FUNCTION_BLOCK PLC01A1 (* Access IOs of the PLC01A1 module *)
  (* Standard: 61499-2; Description: Copyright (c) 2019 fortiss GmbH This program and the accompanying materials are made available under the terms of the Eclipse Public License 2.0 which is available at https://www.eclipse.org/legal/epl-2.0/ SPDX-License-Identifier: EPL-2.0 *)
  (* Version 1.0, 2019-10-01, Jose Cabral, fortiss GmbH *)
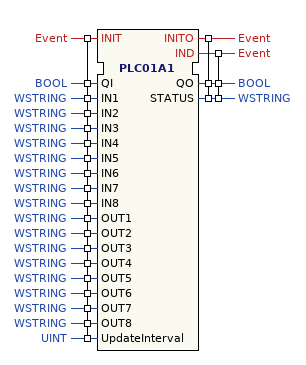
  EVENT_INPUT
    INIT WITH QI, UpdateInterval, IN1, IN2, IN3, IN4, IN5, IN6, IN7, IN8, OUT1, OUT2, OUT3, OUT4, OUT5, OUT6, OUT7, OUT8; (* Service Initialization *)
  END_EVENT
  EVENT_OUTPUT
    INITO WITH QO, STATUS; (* Initialization Confirm *)
    IND WITH QO, STATUS; (* Indication from Resource *)
  END_EVENT
  VAR_INPUT
    QI : BOOL; (* Event Input Qualifier *)
    IN1 : WSTRING;
    IN2 : WSTRING;
    IN3 : WSTRING;
    IN4 : WSTRING;
    IN5 : WSTRING;
    IN6 : WSTRING;
    IN7 : WSTRING;
    IN8 : WSTRING;
    OUT1 : WSTRING;
    OUT2 : WSTRING;
    OUT3 : WSTRING;
    OUT4 : WSTRING;
    OUT5 : WSTRING;
    OUT6 : WSTRING;
    OUT7 : WSTRING;
    OUT8 : WSTRING;
    UpdateInterval : UINT := 25; (* Update interval in Hz *)
  END_VAR
  VAR_OUTPUT
    QO : BOOL; (* Event Output Qualifier *)
    STATUS : WSTRING; (* Service Status *)
  END_VAR
  (* Service APPLICATION/RESOURCE: Access IOs of the PLC01A1 module *)
END_FUNCTION_BLOCK
